# B&R Automation Studio project LyskrydsTA
Automation Studio 4.3.3.196

## Configuration Config1

### Task classes (Cpu.sw)
```
Cyclic#4:
  Program <- Program.prg
VcDataObjects: Visu <- Visu.dob
Libraries: standard
```

### Hardware
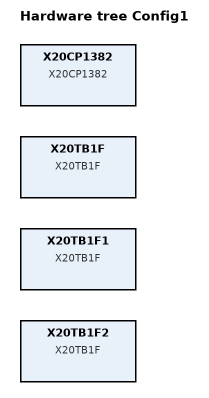
```
X20CP1382 : X20CP1382 v1.3.2.0  [X1 -> X1.SL; X2 -> X2.SL; X3 -> X3.SL]
  Module X1 (Type=X1, Virtual=true, Version=1.3.2.0)
    Connection (Connector=SS1, TargetModule=X20TB1F, TargetConnector=SS)
    Connection (Connector=SL, TargetModule=X20CP1382, TargetConnector=X1)
  Module X2 (Type=X2, Virtual=true, Version=1.3.2.0)
    Connection (Connector=SS1, TargetModule=X20TB1F1, TargetConnector=SS)
    Connection (Connector=SL, TargetModule=X20CP1382, TargetConnector=X2)
  Module X3 (Type=X3, Virtual=true, Version=1.3.2.0)
    Connection (Connector=SS1, TargetModule=X20TB1F2, TargetConnector=SS)
    Connection (Connector=SL, TargetModule=X20CP1382, TargetConnector=X3)
  Connector IF2:
    ActivateDevice = 1
    Vnc1
    VncVcObjectName1 = Visu
    VncKeyMappingFile1 = VC\PS2-Keyboard.dis
  ConfigurationID = LyskrydsTA_Config1
  Simulation = 1
X20TB1F : X20TB1F v1.0.0.0
X20TB1F1 : X20TB1F v1.0.0.0
X20TB1F2 : X20TB1F v1.0.0.0
```

## Logical view

### Program Logical/Program (IEC)

#### Types.typ
```iecst
TYPE
	light_north :
		(
		yellow_north,
		green_north,
		red_north,
		ry_north
		);
	light_west :
		(
		yellow_west,
		green_west,
		red_west
		);
	light_south :
		(
		yellow_south,
		green_south,
		red_south
		);
	light_east :
		(
		yellow_east,
		green_east,
		red_east,
		ry_east
		);
END_TYPE
```

#### Variables.var
```iecst
VAR
	car_from_east : BOOL;
	car_from_north : BOOL;
	car_from_south : BOOL;
	car_from_west : BOOL;
	green_east_bool : BOOL;
	green_north_bool : BOOL;
	green_south_bool : BOOL;
	green_west_bool : BOOL;
	light_state_east : light_east;
	light_state_north : light_north;
	light_state_south : light_south;
	light_state_west : light_west;
	ry_east_bool : BOOL;
	ry_west_bool : BOOL;
	ry_south_bool : BOOL;
	ry_north_bool : BOOL;
	light_timer : TON;
	red_east_bool : BOOL;
	red_north_bool : BOOL;
	red_south_bool : BOOL;
	red_west_bool : BOOL;
	yellow_east_bool : BOOL;
	yellow_north_bool : BOOL;
	yellow_south_bool : BOOL;
	yellow_west_bool : BOOL;
END_VAR
```

#### Main.st
```iecst
PROGRAM _INIT
	(* Insert code here *)
	light_state_north := red_north;
	light_state_east := green_east;
END_PROGRAM

PROGRAM _CYCLIC

	//Timer at 1.5ms for each light change

	CASE light_state_north OF

		red_north:

			light_timer.IN := TRUE;
			light_timer.PT := T#1500ms;

			IF light_timer.Q THEN
				red_north_bool := TRUE;
				red_south_bool := TRUE;
				yellow_south_bool := TRUE;
				yellow_north_bool := TRUE;
				green_north_bool := FALSE;
				green_south_bool := FALSE;
				light_state_north := ry_north;
				light_timer.IN := FALSE;
			END_IF

		yellow_north:

			light_timer.IN := TRUE;
			light_timer.PT := T#1500ms;

			IF light_timer.Q THEN
				red_north_bool := FALSE;
				red_south_bool := FALSE;
				yellow_north_bool := FALSE;
				yellow_south_bool := FALSE;
				green_south_bool := TRUE;
				green_north_bool := TRUE;
				light_state_north := green_north;
				light_timer.IN := FALSE;
			END_IF

		green_north:

			light_timer.IN := TRUE;
			light_timer.PT := T#1500ms;

			IF light_timer.Q THEN
				red_north_bool := FALSE;
				red_south_bool := FALSE;
				yellow_north_bool := TRUE;
				yellow_south_bool := TRUE;
				green_south_bool := FALSE;
				green_north_bool := FALSE;
				light_state_north := yellow_north;
				light_timer.IN := FALSE;
			END_IF

		ry_north:

			light_timer.IN := TRUE;
			light_timer.PT := T#1500ms;

			IF light_timer.Q THEN
				red_north_bool := FALSE;
				red_south_bool := FALSE;
				yellow_north_bool := FALSE;
				yellow_south_bool := FALSE;
				green_south_bool := TRUE;
				green_north_bool := TRUE;
				light_state_north := green_north;
				light_timer.IN := FALSE;
			END_IF

	END_CASE

	CASE light_state_east OF

		red_east:

			light_timer.IN := TRUE;
			light_timer.PT := T#1500ms;

			IF light_timer.Q THEN
				red_west_bool := TRUE;
				red_east_bool := TRUE;
				yellow_west_bool := TRUE;
				yellow_east_bool := TRUE;
				light_state_east := yellow_east;
				light_timer.IN := FALSE;
			END_IF

		yellow_east:
			light_timer.IN := TRUE;
			light_timer.PT := T#1500ms;

			IF light_timer.Q THEN
				red_west_bool := FALSE;
				red_east_bool := FALSE;
				yellow_west_bool := FALSE;
				yellow_east_bool := FALSE;
				green_west_bool := TRUE;
				green_east_bool := TRUE;
				light_state_east := green_east;
				light_timer.IN := FALSE;
			END_IF
		green_east:

			light_timer.IN := TRUE;
			light_timer.PT := T#1500ms;

			IF light_timer.Q THEN
				red_west_bool := FALSE;
				red_east_bool := FALSE;
				yellow_west_bool := TRUE;
				yellow_east_bool := TRUE;
				green_west_bool := FALSE;
				green_east_bool := FALSE;
				light_state_east := yellow_east;
				light_timer.IN := FALSE;
			END_IF

		ry_east:

			light_timer.IN := TRUE;
			light_timer.PT := T#1500ms;

			IF light_timer.Q THEN
				red_west_bool := FALSE;
				red_east_bool := FALSE;
				yellow_west_bool := FALSE;
				yellow_east_bool := FALSE;
				green_west_bool := TRUE;
				green_east_bool := TRUE;
				light_state_east := green_east;
				light_timer.IN := FALSE;
			END_IF

	END_CASE

	light_timer();

END_PROGRAM

PROGRAM _EXIT
	(* Insert code here *)

END_PROGRAM
```

- Visualisation Logical/Visu (not shown)

Listed in the project but not available here: Logical/Global.typ, Logical/Global.var, Logical/Libraries
